// TIA Portal V21 export
DATA_BLOCK "数据块_2"   // DB3
{ S7_Optimized_Access := 'TRUE' }
// stored: AutoNumber false, MemoryReserve 100
   VAR
      cntDb : DInt;
   END_VAR
BEGIN
END_DATA_BLOCK
